// TwinCAT 3 PLC project Untitled1
// ProgramVersion: 3.1.4023.0
// libraries:
//   Tc2_Standard, * (Beckhoff Automation GmbH)
//   Tc2_System, * (Beckhoff Automation GmbH)
//   Tc2_Utilities, * (Beckhoff Automation GmbH)
//   Tc3_IotBase, * (Beckhoff Automation GmbH)
//   Tc3_Module, * (Beckhoff Automation GmbH)
// project tree:
//   DUTs/ MQTTSettings.TcDUT (not stored)
//   / PlcTask.TcTTO
//   POUs/ MAIN.TcPOU, MQTT.TcPOU, MQTTTest.TcPOU, Servo.TcPOU
// real-time tasks:
//   TASK PlcTask: cycle T#10ms, priority 20, ADS port 350

CONFIGURATION Untitled1
    RESOURCE PLC ON TwinCAT3
        TASK PlcTask(INTERVAL := T#10ms, PRIORITY := 20);
        PROGRAM MAIN WITH PlcTask : MAIN;
    END_RESOURCE
END_CONFIGURATION

// ---- POUs/MAIN.TcPOU
PROGRAM MAIN
VAR
	mqtt: MQTT;
	//mqttTest: MQTTTest;

	angleTimer : TON := (PT:=T#1S);
	speedTimer : TON := (PT:=T#10MS);
	tonTimerCounter : TON := (PT:=T#100MS);
	tonTimerMessage : TON := (PT:=T#100MS);
	
	servo : Servo;
	angle : INT;
	
END_VAR

IF _TaskInfo[GETCURTASKINDEXEX()].FirstCycle THEN
	mqtt.configureMQTTClient();
END_IF 
mqtt.connect();

servo.waitForCommand(mqtt := mqtt);
servo.publishAngle(mqtt := mqtt, timer := angleTimer);
servo.publishSpeed(mqtt := mqtt, timer := speedTimer);

//mqttTest.counterTest(tonTimer:=tonTimerCounter, mqtt:=mqtt);
//mqttTest.messageTest(tonTimer:=tonTimerMessage, mqtt:=mqtt, msg:='some fixed msg');
//mqttTest.capacityTest(mqtt:=mqtt);

END_PROGRAM

// ---- POUs/MQTT.TcPOU
FUNCTION_BLOCK MQTT
VAR_OUTPUT
	mqttClient : FB_IotMqttClient;
END_VAR
VAR
	mqttSettings : MQTTSettings;
	messageQueue : FB_IotMqttMessageQueue;
    message      : FB_IotMqttMessage;
	isSubscribed : BOOL;
	
	counterTestTopic : STRING := 'plc/counterTest';
	messageTestTopic : STRING := 'plc/messageTest';
	capacityTestTopic : STRING := 'plc/capacityTest';
	
	counter : INT := 0;
END_VAR

METHOD PUBLIC configureMQTTClient
VAR_IN_OUT
END_VAR
mqttClient.sHostName := mqttSettings.brokerIP;
mqttClient.nHostPort := mqttSettings.brokerPort;
mqttClient.sClientId := mqttSettings.clientId;
mqttClient.sUserName := mqttSettings.brokerUsername;
mqttClient.sUserPassword := mqttSettings.brokerPassword;
mqttClient.stTLS.sCA := mqttSettings.caCertificateAbsolutePath;
mqttClient.stTLS.sCert := mqttSettings.clientCertificateAbsolutePath;
mqttClient.stTLS.sKeyFile := mqttSettings.clientKeyAbsolutePath;
mqttClient.ipMessageQueue := messageQueue;
END_METHOD

METHOD PUBLIC connect
mqttClient.Execute(bConnect := TRUE);
END_METHOD

METHOD PUBLIC isConnected : BOOL
isConnected := mqttClient.bConnected;
END_METHOD

METHOD PUBLIC publish : BOOL
VAR_INPUT
	msg : STRING;
END_VAR
mqttClient.Publish(sTopic:= mqttSettings.topicPub,
            pPayload:= ADR(msg),
            nPayloadSize:= LEN2(ADR(msg))+1,
            eQoS:= mqttSettings.qos,
            bRetain:= FALSE,
            bQueue:= FALSE
);
END_METHOD

METHOD publishBack : BOOL
VAR_INPUT
END_VAR
VAR
	receivedTopic : STRING(255);
	receivedMsg : STRING(255);
END_VAR
IF isConnected() THEN
	IF NOT isSubscribed THEN
        isSubscribed := mqttClient.Subscribe(sTopic:=mqttSettings.topicSub, eQoS:=mqttSettings.qos);
    END_IF	

	IF messageQueue.nQueuedMessages > 0 THEN	
		IF messageQueue.Dequeue(fbMessage:=message) THEN
			message.GetTopic(pTopic:=ADR(receivedTopic), nTopicSize:=SIZEOF(receivedTopic) );
			message.GetPayload(pPayload:=ADR(receivedMsg), nPayloadSize:=SIZEOF(receivedMsg), bSetNullTermination:=FALSE);

			publish(msg := receivedMsg);
		END_IF
	END_IF
	
END_IF
END_METHOD

METHOD PUBLIC publishToTopic : BOOL
VAR_INPUT
	topic : STRING;
	msg : STRING;
END_VAR
mqttClient.Publish(sTopic:= topic,
            pPayload:= ADR(msg),
            nPayloadSize:= LEN2(ADR(msg))+1,
            eQoS:= mqttSettings.qos,
            bRetain:= FALSE,
            bQueue:= FALSE
);
END_METHOD

METHOD PUBLIC publishWithTON
VAR_IN_OUT
	timer : TON;	
END_VAR
VAR_INPUT
	msg : STRING;
END_VAR
IF isConnected() THEN
    timer(IN:=TRUE);
    IF timer.Q THEN
        timer(IN:=FALSE);
     
        publish(msg := msg);
    END_IF
END_IF
END_METHOD

END_FUNCTION_BLOCK

// ---- POUs/Servo.TcPOU
FUNCTION_BLOCK Servo
VAR
	mqttSettings : MQTTSettings;	

	currentSpeed : INT;
	currentAngle : INT;
	
	servoAngleCommandTopic : STRING := 'plc/servo/angle';
	servoAngleOutTopic : STRING := 'plc/servo/angle/out';
	servoSpeedOutTopic : STRING := 'plc/servo/speed/out';
	isSubscribed : BOOL := FALSE;
END_VAR

METHOD getAngle : INT
VAR_OUTPUT
	angle : INT;
END_VAR
angle := currentAngle;
END_METHOD

METHOD publishAngle
VAR_IN_OUT
	mqtt: MQTT;	
	timer : TON;
END_VAR
IF mqtt.isConnected() THEN
    timer(IN:=TRUE);
    IF timer.Q THEN
        timer(IN:=FALSE);
        mqtt.publishToTopic(topic := servoAngleOutTopic, msg := INT_TO_STRING(currentAngle));
    END_IF
END_IF
END_METHOD

METHOD publishSpeed
VAR_IN_OUT
	mqtt: MQTT;	
	timer : TON;
END_VAR
IF mqtt.isConnected() THEN
    timer(IN:=TRUE);
    IF timer.Q THEN
        timer(IN:=FALSE);
        mqtt.publishToTopic(topic := servoSpeedOutTopic, msg := INT_TO_STRING(currentSpeed));
    END_IF
END_IF
END_METHOD

METHOD setAngle : BOOL
VAR_INPUT
	angleToSet : INT;
END_VAR
currentAngle := angleToSet;
END_METHOD

METHOD waitForCommand
VAR_IN_OUT
	mqtt: MQTT;	
END_VAR
VAR
	receivedMsg : STRING(255);
	
	angleToSet : INT;
END_VAR
IF mqtt.isConnected() THEN
	IF NOT isSubscribed THEN
        isSubscribed := mqtt.mqttClient.Subscribe(sTopic:=servoAngleCommandTopic, eQoS:=mqttSettings.qos);
    END_IF	

	IF mqtt.messageQueue.nQueuedMessages > 0 THEN	
		IF mqtt.messageQueue.Dequeue(fbMessage:=mqtt.message) THEN
			IF mqtt.message.CompareTopic(sTopic:=servoAngleCommandTopic) THEN	
	
				mqtt.message.GetPayload(pPayload:=ADR(receivedMsg), nPayloadSize:=SIZEOF(receivedMsg), bSetNullTermination:=FALSE);				
				angleToSet := STRING_TO_INT(receivedMsg);
				IF (angleToSet >= 0 AND angleToSet <= 360) THEN
					setAngle(angleToSet := angleToSet);
				END_IF
			
			END_IF
		END_IF
	END_IF
	
END_IF
END_METHOD

END_FUNCTION_BLOCK

// ---- POUs/MQTTTest.TcPOU
FUNCTION_BLOCK MQTTTest
VAR_INPUT
END_VAR
VAR_OUTPUT
END_VAR
VAR
	mqttSettings : MQTTSettings;

	counterTestTopic : STRING := 'plc/counterTest';
	messageTestTopic : STRING := 'plc/messageTest';
	capacityTestTopic : STRING := 'plc/capacityTest';
	
	counter : INT := 0;
	isSubscribed : BOOL := false;
END_VAR

METHOD capacityTest : BOOL
VAR_IN_OUT
	mqtt: MQTT;	
END_VAR
VAR
	receivedMsg : STRING(255);
END_VAR
IF mqtt.isConnected() THEN
	IF NOT isSubscribed THEN
        isSubscribed := mqtt.mqttClient.Subscribe(sTopic:=capacityTestTopic, eQoS:=mqttSettings.qos);
    END_IF	

	IF mqtt.messageQueue.nQueuedMessages > 0 THEN	
		IF mqtt.messageQueue.Dequeue(fbMessage:=mqtt.message) THEN
			IF mqtt.message.CompareTopic(sTopic:=capacityTestTopic) THEN	
	
				mqtt.message.GetPayload(pPayload:=ADR(receivedMsg), nPayloadSize:=SIZEOF(receivedMsg), bSetNullTermination:=FALSE);				
				mqtt.publishToTopic(topic:=CONCAT(capacityTestTopic, '/out'), msg := receivedMsg);
			
			END_IF
		END_IF
	END_IF
	
END_IF
END_METHOD

METHOD PUBLIC counterTest
VAR_IN_OUT
	tonTimer : TON;
	mqtt: MQTT;	
END_VAR
IF mqtt.isConnected() THEN
	tonTimer(IN:=TRUE);
	IF tonTimer.Q THEN
		tonTimer(IN:=FALSE);
		counter := counter + 1;			  
		mqtt.publishToTopic(msg:=TO_STRING(counter), topic:=counterTestTopic);
	END_IF
END_IF
END_METHOD

METHOD messageTest : BOOL
VAR_IN_OUT
	tonTimer : TON;
	mqtt : MQTT;	
	
END_VAR
VAR_INPUT
	msg : STRING;
END_VAR
IF mqtt.isConnected() THEN	
	
    tonTimer(IN:=TRUE);
    IF tonTimer.Q THEN
		mqtt.publishToTopic(msg:=msg, topic:=messageTestTopic);			
        tonTimer(IN:=FALSE);  
    END_IF
	
END_IF
END_METHOD

END_FUNCTION_BLOCK
